{attribute addProperty BoxType "EP9128-0021-0019"}
{attribute addProperty Id "A_0016_EP9214_0023_0019EP9214_FC34E2BF62678.25A_0017_EP9214_0023_0020EP9214_FC34E2BF62678.25A_0018_EP9214_0023_0021EP9214_FC34E2BF62678.25A_0019_EP9214_0023_0022EP9214_FC34E2BF62678.25A_0020_EP9224_0023_0016EP9224_D133F73C882110.25A_0021_EP9224_0023_0017EP9224_D133F73C882110.25A_0024_EP9521_0020_0000A_0024_EP9521_0020_0000_2C408F2A21827.25A_0022_EP9224_0037_0017A_0022_EP9224_0037_0017_E33DE408162A_0013_EP9128_0021_0019_2_EP9128_1021EP9128_179A0949162A_0013_EP9128_0021_0019_3_EP9128_2021EP9128_179A0949162"}
{attribute addProperty CRC "133026282"}
{attribute addProperty SizeInBites "4534"}
{attribute addProperty SizeInBytes "566.75"}
TYPE A_0013_EP9128_0021_0019_07EDD1EA EXTENDS EP9128_179A0949 :
STRUCT
	{attribute addProperty Name "A_0016_EP9214_0023_0019"}
	A_0016_EP9214_0023_0019 : EP9214_FC34E2BF;
	{attribute addProperty Name "A_0017_EP9214_0023_0020"}
	A_0017_EP9214_0023_0020 : EP9214_FC34E2BF;
	{attribute addProperty Name "A_0018_EP9214_0023_0021"}
	A_0018_EP9214_0023_0021 : EP9214_FC34E2BF;
	{attribute addProperty Name "A_0019_EP9214_0023_0022"}
	A_0019_EP9214_0023_0022 : EP9214_FC34E2BF;
	{attribute addProperty Name "A_0020_EP9224_0023_0016"}
	A_0020_EP9224_0023_0016 : EP9224_D133F73C;
	{attribute addProperty Name "A_0021_EP9224_0023_0017"}
	A_0021_EP9224_0023_0017 : EP9224_D133F73C;
	{attribute addProperty Name "A_0024_EP9521_0020_0000"}
	A_0024_EP9521_0020_0000 : A_0024_EP9521_0020_0000_2C408F2A;
	{attribute addProperty Name "A_0022_EP9224_0037_0017"}
	A_0022_EP9224_0037_0017 : A_0022_EP9224_0037_0017_E33DE408;
	{attribute addProperty Name "A_0013_EP9128_0021_0019_2_EP9128_1021"}
	A_0013_EP9128_0021_0019_2_EP9128_1021 : EP9128_179A0949;
	{attribute addProperty Name "A_0013_EP9128_0021_0019_3_EP9128_2021"}
	A_0013_EP9128_0021_0019_3_EP9128_2021 : EP9128_179A0949;
END_STRUCT
END_TYPE

(* stored: Version 1.2.0.0, ProductVersion 3.1.4024.9
   DUT A_0013_EP9128_0021_0019_07EDD1EA: Id {824c7ffb-cd04-46da-9d5e-5ee6d758debb} *)
